FUNCTION_BLOCK RT_E_DEMUX (* Event demultiplexer *)
  (* Description: Copyright (c) 2008 ACIN This program and the accompanying materials are made available under the terms of the Eclipse Public License 2.0 which is available at https://www.eclipse.org/legal/epl-2.0/ SPDX-License-Identifier: EPL-2.0 *)
  (* Version 3.0, 2025-04-14, Patrick Aigner, changed package *)
  (* Version 1.0, 2008-07-10, Alois Zoitl, ACIN *)
  PACKAGE eclipse4diac::rtevents;
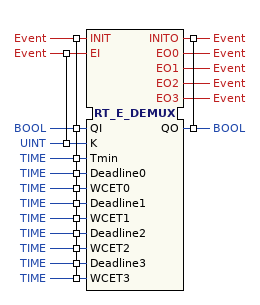
  EVENT_INPUT
    INIT WITH QI, Tmin, Deadline0, WCET0, Deadline1, WCET1, Deadline2, WCET2, Deadline3, WCET3;
    EI WITH K; (* Event to demultiplex *)
  END_EVENT
  EVENT_OUTPUT
    INITO WITH QO;
    EO0;
    EO1;
    EO2;
    EO3; (* Number of outputs is implementation dependent *)
  END_EVENT
  VAR_INPUT
    QI : BOOL;
    K : UINT; (* Event index,maximum is implementation dependent *)
    Tmin : TIME;
    Deadline0 : TIME;
    WCET0 : TIME;
    Deadline1 : TIME;
    WCET1 : TIME;
    Deadline2 : TIME;
    WCET2 : TIME;
    Deadline3 : TIME;
    WCET3 : TIME;
  END_VAR
  VAR_OUTPUT
    QO : BOOL;
  END_VAR
END_FUNCTION_BLOCK
